# EPICS substitutions: op-m3b/6POD/db/6Pod_DigitalChannels.substitutions
file db/SAI_DigitalChannels.template {
pattern {	P,		R,		SCAN, 		ASYNPORT}
        { 	"XF:23ID2-OP","{Mir:3B}",	"1 second",	"pmac"}
}

# Sample Naming - XF:23ID2-OP{Mir:3B-Ax:1}Mtr
#EOF
